FUNCTION_BLOCK FB_MotionAxisNC IMPLEMENTS I_MotionAxis
VAR CONSTANT
    nOFFSET_TO_PLCTONC_AXIS_REF_CTRL : LWORD := 0;
END_VAR
VAR
    AxisReference : REFERENCE TO AXIS_REF;

    AxisReference_PLCtoNC_ControlDWord : MC.PLCTONC_AXIS_REF_CTRL;

    fbMcReset : MC_Reset;
    fbMcPower : MC_Power;

    fbMcMoveAbsolute : MC_MoveAbsolute;

    bMostRecentMoveAbsoluteDone : BOOL;
END_VAR


AxisReference.ReadStatus();

MEMCPY(
    ADR(AxisReference_PLCtoNC_ControlDWord),
    ADR(AxisReference.PlcToNc) + nOFFSET_TO_PLCTONC_AXIS_REF_CTRL,
    SIZEOF(AxisReference_PLCtoNC_ControlDWord)
);

fbMcReset(
    Axis := AxisReference,
    Execute := FALSE
);

fbMcPower(Axis := AxisReference);

fbMcMoveAbsolute(
    Axis := AxisReference,
    Execute := FALSE
);

IF THIS^.fbMcMoveAbsolute.Done THEN
    THIS^.bMostRecentMoveAbsoluteDone := TRUE;
END_IF


METHOD FB_Init: BOOL
VAR_INPUT
    bInitRetains: BOOL; // TRUE: the retain variables are initialized (reset warm / reset cold)
    bInCopyCode: BOOL;  // TRUE: the instance will be copied to the copy code afterward (online change)

    AxisReference : REFERENCE TO AXIS_REF;
    MotionInterlock : I_MotionInterlock;
    MotionAxisMoveAbsolute : I_MotionAxisMoveAbsolute;
    MotionAxisHome : I_MotionAxisHome;
    MotionAxisReset : I_MotionAxisReset;
END_VAR

THIS^.AxisReference REF= AxisReference;
THIS^.iMotionAxisMoveAbsolute := MotionAxisMoveAbsolute;
END_METHOD


METHOD GetAxisRef : REFERENCE TO AXIS_REF

GetAxisRef REF= THIS^.AxisReference;
END_METHOD


METHOD GetPowerOverride : LREAL

GetPowerOverride := TO_LREAL(THIS^.AxisReference.PlcToNc.Override) / 10000.0;
END_METHOD

{warning 'Add method implementation '}
METHOD Home
END_METHOD

{warning 'Add property implementation'}
PROPERTY MeasuredAcceleration : LREAL
GET

MeasuredAcceleration := THIS^.AxisReference.NcToPlc.ActAcc;
END_GET
END_PROPERTY

{warning 'Add property implementation'}
PROPERTY MeasuredPosition : LREAL
GET

MeasuredPosition := THIS^.AxisReference.NcToPlc.ActPos;
END_GET
END_PROPERTY

{warning 'Add property implementation'}
PROPERTY MeasuredVelocity : LREAL
GET

MeasuredVelocity := THIS^.AxisReference.NcToPlc.ActVelo;
END_GET
END_PROPERTY


METHOD MoveAbsolute
VAR_INPUT
    Position	: LREAL;
    Velocity	: LREAL;
    Acceleration	: LREAL := 0.0;
    Deceleration	: LREAL := 0.0;
    Jerk	: LREAL := 0.0;
    BufferMode	: MC_BufferMode := MC_BufferMode.MC_Aborting;
END_VAR
VAR_OUTPUT
    Done	: BOOL;
    Busy	: BOOL;
    Active	: BOOL;
    CommandAborted	: BOOL;
    Error	: BOOL;
    ErrorID	: UDINT;
    ErrorStr	: T_MaxString;
END_VAR

bMostRecentMoveAbsoluteDone := FALSE;

THIS^.fbMcMoveAbsolute(
    Axis := THIS^.AxisReference,
    Execute := TRUE,
    Position := Position,
    Velocity := Velocity,
    Acceleration := Acceleration,
    Deceleration := Deceleration,
    Jerk := Jerk,
    BufferMode := BufferMode,
    Done => Done,
    Busy => Busy,
    Active => Active,
    CommandAborted => CommandAborted,
    Error => Error,
    ErrorID => ErrorID
);

ErrorStr := '';
END_METHOD


PROPERTY MoveAbsoluteBusy : BOOL
GET

MoveAbsoluteBusy := THIS^.fbMcMoveAbsolute.Busy;
END_GET
END_PROPERTY


PROPERTY MoveAbsoluteDone : BOOL
GET

MoveAbsoluteDone := THIS^.fbMcMoveAbsolute.Done OR THIS^.bMostRecentMoveAbsoluteDone;
END_GET
END_PROPERTY


PROPERTY MoveAbsoluteError : BOOL
GET

MoveAbsoluteError := THIS^.fbMcMoveAbsolute.Error;
END_GET
END_PROPERTY


PROPERTY MoveAbsoluteErrorID : UDINT
GET

MoveAbsoluteErrorID := THIS^.fbMcMoveAbsolute.ErrorID;
END_GET
END_PROPERTY

{warning 'Add property implementation'}
PROPERTY MoveAbsoluteTargetAcceleration : LREAL
GET

MoveAbsoluteTargetAcceleration := THIS^.fbMcMoveAbsolute.Acceleration;
END_GET
END_PROPERTY

{warning 'Add property implementation'}
PROPERTY MoveAbsoluteTargetDeceleration : LREAL
GET

MoveAbsoluteTargetDeceleration := THIS^.fbMcMoveAbsolute.Deceleration;
END_GET
END_PROPERTY

{warning 'Add property implementation'}
PROPERTY MoveAbsoluteTargetJerk : LREAL
GET

MoveAbsoluteTargetJerk := THIS^.fbMcMoveAbsolute.Jerk;
END_GET
END_PROPERTY

{warning 'Add property implementation'}
PROPERTY MoveAbsoluteTargetPosition : LREAL
GET

MoveAbsoluteTargetPosition := THIS^.fbMcMoveAbsolute.Position;
END_GET
END_PROPERTY

{warning 'Add property implementation'}
PROPERTY MoveAbsoluteTargetVelocity : LREAL
GET

MoveAbsoluteTargetVelocity := THIS^.fbMcMoveAbsolute.Velocity;
END_GET
END_PROPERTY


PROPERTY NegativeMotionIsEnabled : BOOL
GET

NegativeMotionIsEnabled := THIS^.AxisReference_PLCtoNC_ControlDWord.2;;
END_GET
END_PROPERTY


PROPERTY PositiveMotionIsEnabled : BOOL
GET

PositiveMotionIsEnabled := THIS^.AxisReference_PLCtoNC_ControlDWord.1;
END_GET
END_PROPERTY


METHOD Power
VAR_INPUT
    Enable	: BOOL;
    Enable_Positive	: BOOL;
    Enable_Negative	: BOOL;
    (* in percent from 0 to 100 *)
    Override	: LREAL := 100.0;
    BufferMode	: MC_BufferMode := MC_BufferMode.MC_Aborting;
END_VAR
VAR_OUTPUT
    Status	: BOOL;
    Busy	: BOOL;
    Active	: BOOL;
    Error	: BOOL;
    ErrorID	: UDINT;
    ErrorStr	: T_MaxString;
END_VAR

THIS^.fbMcPower(
    Axis := THIS^.AxisReference,
    Enable := Enable,
    Enable_Positive := Enable_Positive,
    Enable_Negative := Enable_Negative,
    Override := Override,
    BufferMode := BufferMode,
    Status => Status,
    Busy => Busy,
    Active => Active,
    Error => Error,
    ErrorID => ErrorID
);

ErrorStr := '';
END_METHOD


PROPERTY PowerError : BOOL
GET

PowerError := THIS^.fbMcPower.Error;
END_GET
END_PROPERTY


PROPERTY PowerErrorID : UDINT
GET

PowerErrorID := THIS^.fbMcPower.ErrorID;
END_GET
END_PROPERTY

{warning 'Add method implementation '}
METHOD PowerErrorIDToStr : T_MaxString
VAR_INPUT
    ErrorID : UDINT;
END_VAR
END_METHOD


PROPERTY PowerIsEnabled : BOOL
GET

PowerIsEnabled := THIS^.AxisReference_PLCtoNC_ControlDWord.0;
END_GET
END_PROPERTY


PROPERTY PowerOverride : LREAL
GET

PowerOverride := GetPowerOverride();
END_GET
END_PROPERTY


PROPERTY PowerStatus : BOOL
GET

PowerStatus := THIS^.fbMcPower.Status;
END_GET
END_PROPERTY


METHOD Reset
VAR_OUTPUT
    Done : BOOL;
    Busy : BOOL;
    Error : BOOL;
    ErrorID : UDINT;
    ErrorStr : T_MaxString;
END_VAR

THIS^.fbMcReset(
    Axis := THIS^.AxisReference,
    Execute := TRUE,
    Done => Done,
    Busy => Busy,
    Error => Error,
    ErrorID => ErrorID,
);

ErrorStr := '';
END_METHOD

{warning 'Add property implementation'}
PROPERTY SetpointAcceleration : LREAL
GET

SetpointAcceleration := THIS^.AxisReference.NcToPlc.SetAcc;
END_GET
END_PROPERTY

{warning 'Add property implementation'}
PROPERTY SetpointJerk : LREAL
GET

SetpointJerk := THIS^.AxisReference.NcToPlc.SetJerk;
END_GET
END_PROPERTY

{warning 'Add property implementation'}
PROPERTY SetpointPosition : LREAL
GET

SetpointPosition := THIS^.AxisReference.NcToPlc.SetPos;
END_GET
END_PROPERTY

{warning 'Add property implementation'}
PROPERTY SetpointVelocity : LREAL
GET

SetpointVelocity := THIS^.AxisReference.NcToPlc.SetVelo;
END_GET
END_PROPERTY


METHOD SetPowerOverride
VAR_INPUT
    (* in percent from 0 to 100 *)
    Override	: LREAL;
END_VAR
VAR_OUTPUT
    Status	: BOOL;
    Busy	: BOOL;
    Active	: BOOL;
    Error	: BOOL;
    ErrorID	: UDINT;
    ErrorStr	: T_MaxString;
END_VAR

THIS^.fbMcPower(
    Axis := THIS^.AxisReference,
    Override := Override,
    Status => Status,
    Busy => Busy,
    Error => Error,
    ErrorID => ErrorID
);

ErrorStr := '';
END_METHOD

END_FUNCTION_BLOCK

(* stored: Version 1.1.0.1
   POU FB_MotionAxisNC: Id {9be303f4-acd5-4745-885a-80a353f6baa1}, SpecialFunc None
   Method FB_Init: Id {546afd61-8f00-40dc-8d41-5f7ef58b9805}
   Method GetAxisRef: Id {b97afe87-af3e-48e5-ad17-4f33de4e42d3}
   Method GetPowerOverride: Id {70e762d0-7e7f-4eac-be4f-cd33c65d3e2e}
   Method Home: Id {442d628d-e7c2-4655-926e-f3676b5bfba8}
   Property MeasuredAcceleration: Id {ce700626-182a-451d-9661-33afae0932de}
   Get Get: Id {24638d8d-4f8c-4764-b353-b63ee014a191}
   Property MeasuredPosition: Id {d3c3156d-ba89-48d7-91f8-4e7a165cc66b}
   Get Get: Id {6386dbc4-f87a-4181-bddc-a0cc57582702}
   Property MeasuredVelocity: Id {a1b1d885-c261-4693-b29c-e39d15a3b486}
   Get Get: Id {38c3a806-cf80-4d8d-ac8f-1f20820ef064}
   Method MoveAbsolute: Id {ee6574eb-b826-4f9c-9a4d-d9a7fbacdb97}
   Property MoveAbsoluteBusy: Id {aa611738-39cc-4180-b661-628ea72244af}
   Get Get: Id {76e43a73-b711-4837-8c2c-e03c439d6822}
   Property MoveAbsoluteDone: Id {7a171aa6-c700-4c1a-b567-d53853a5e431}
   Get Get: Id {31360ced-32cd-4b5d-9660-4df4da302b78}
   Property MoveAbsoluteError: Id {1177e88e-776d-4083-860e-fe1ac9d94cb0}
   Get Get: Id {9310b682-078b-4e02-b576-b03dd2cccc90}
   Property MoveAbsoluteErrorID: Id {a1c09038-1afa-4065-b167-41bacd8c3d62}
   Get Get: Id {eb80a200-a7fe-4701-86c3-01b5d3d386c7}
   Property MoveAbsoluteTargetAcceleration: Id {5683ee99-a7cb-40c2-969a-a474cbabb860}
   Get Get: Id {74ac094b-307f-4b5f-91ca-d6df23e4b535}
   Property MoveAbsoluteTargetDeceleration: Id {5335ef81-4824-4cb1-8888-7478be067cd1}
   Get Get: Id {40590e54-4383-4bbb-9b93-9becd058e1a3}
   Property MoveAbsoluteTargetJerk: Id {404936f9-3f27-4d57-b379-404e0a170d38}
   Get Get: Id {f2d097b2-7054-4aaf-8d01-6b3c6e222f8d}
   Property MoveAbsoluteTargetPosition: Id {4a5b3ee3-3b45-4442-bac2-ab373b3d1e10}
   Get Get: Id {913c0c9e-9d87-410d-b7bc-77ed2f94846b}
   Property MoveAbsoluteTargetVelocity: Id {a8d7529d-7885-4764-b208-b6ee34051c86}
   Get Get: Id {56022e9f-2342-4dee-bd4b-2a7336c5faab}
   Property NegativeMotionIsEnabled: Id {f929decd-53ae-4f45-bdf0-8fd5a7388369}
   Get Get: Id {dc2bcb41-6866-4082-8722-0da985317d7a}
   Property PositiveMotionIsEnabled: Id {38a8f3fb-b5cf-4671-a122-5f5aa0fe78aa}
   Get Get: Id {32b4a476-1231-40dd-9e5f-7b098fdc6c7a}
   Method Power: Id {a9cc804d-b3dc-434c-baa6-bfc9abd247df}
   Property PowerError: Id {3e15f376-7bf5-4e06-affb-4313d24a4142}
   Get Get: Id {f840f5c8-2446-44e7-8227-7fa75934c87c}
   Property PowerErrorID: Id {75d631eb-9c24-4f0d-8b98-81f2b0ee551c}
   Get Get: Id {453d8769-ae65-4710-93f3-3ed95ffb2240}
   Method PowerErrorIDToStr: Id {e5c2cbc9-22f1-4f8e-8331-1715583bfa7f}
   Property PowerIsEnabled: Id {4195b028-93a8-4321-b9b3-e414b9da8543}
   Get Get: Id {67fde484-f87d-4000-bdd0-312fcc30078f}
   Property PowerOverride: Id {193eb5f4-dd7b-4f3c-80f9-73a98416bf9d}
   Get Get: Id {7a534a31-10a2-4ade-a268-2366bd0172cc}
   Property PowerStatus: Id {0f4d6339-c71d-4d4d-8f69-fea9c613e9c3}
   Get Get: Id {f699dfea-91f3-4196-bb11-bba06d62849a}
   Method Reset: Id {593c499e-31ce-48cf-9b79-08e6bb6550d7}
   Property SetpointAcceleration: Id {e293e00a-7c56-47b2-83d3-ef8933dece0f}
   Get Get: Id {158b8fb5-9724-4d4b-8a6e-15c453f3d6e5}
   Property SetpointJerk: Id {2c243e2e-b1d1-4191-b5c4-cad20400e58c}
   Get Get: Id {4959b303-be94-4c42-a534-68b58ffd8aa4}
   Property SetpointPosition: Id {e45f8292-1580-4ccf-8b4f-96b350c3ad26}
   Get Get: Id {e69de46c-b397-4078-bf83-f3217ab80c4c}
   Property SetpointVelocity: Id {9da29ec4-4354-4699-9043-c2e402c21970}
   Get Get: Id {e115c644-8d6c-4f5c-84de-34bead1ebf46}
   Method SetPowerOverride: Id {93096ca5-9cbe-40de-89ec-d49d761ee091} *)
